PROGRAM CounterUP
VAR

END_VAR

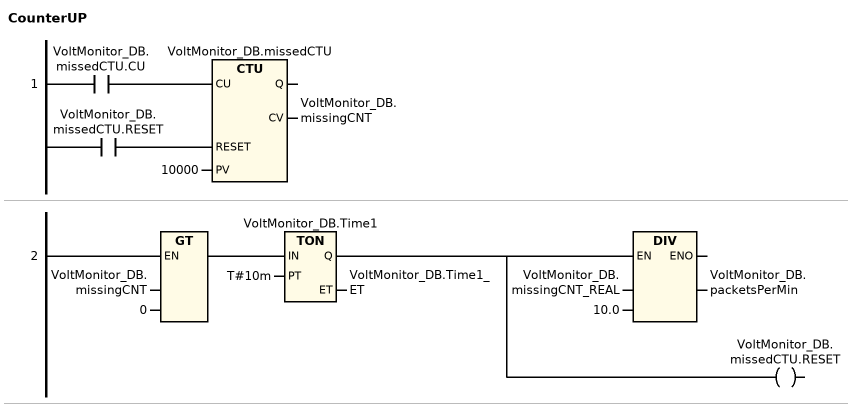
// NETWORK 1
VoltMonitor_DB.missedCTU(
    CU := VoltMonitor_DB.missedCTU.CU,
    RESET := VoltMonitor_DB.missedCTU.RESET,
    PV := 10000,
    CV => VoltMonitor_DB.missingCNT); // CTU

// NETWORK 2
VoltMonitor_DB.Time1(IN := VoltMonitor_DB.missingCNT > 0, PT := T#10m, ET => VoltMonitor_DB.Time1_ET); // TON
IF VoltMonitor_DB.Time1.Q THEN VoltMonitor_DB.packetsPerMin := VoltMonitor_DB.missingCNT_REAL / 10.0; END_IF
VoltMonitor_DB.missedCTU.RESET := VoltMonitor_DB.Time1.Q;

END_PROGRAM

(* stored: Version 1.1.0.1, ProductVersion 3.1.4024.9
   POU CounterUP: Id {163e4b13-2c6a-43c8-9af1-79430eef4cb1}, SpecialFunc None *)
